// TIA Portal V18 export
VAR_GLOBAL   // PLC tag table "MemoryType"
   "PBB Off Mode" AT %M200.0 : Bool;
   "PBB On Mode" AT %M200.1 : Bool;
   "PBB Auto Mode" AT %M200.2 : Bool;
   "Emergency Stop Button Pressed" AT %M200.3 : Bool;
   "Tunnel FW Em Stop LS M" AT %M200.4 : Bool;
   "Tunnel BW Em Stop LS M" AT %M200.5 : Bool;
   "Start M" AT %M200.6 : Bool;
   "Fuse Problem Major" AT %M200.7 : Bool;
   "AutoLeveller Fault" AT %M201.0 : Bool;
   "AutoLeveller Up Over Work" AT %M201.1 : Bool;
   "AutoLeveller Down Over Work" AT %M201.2 : Bool;
   "Driver Error Left" AT %M201.3 : Bool;
   "Driver Error Right" AT %M201.4 : Bool;
   "Wheel Drivers Fault" AT %M201.5 : Bool;
   "SafetyShoe Siren&Info" AT %M201.6 : Bool;
   "SafetyBarrier Activated" AT %M201.7 : Bool;
   "Fault Occurred Major" AT %M202.1 : Bool;
   "Cabin Motor Driver Fault" AT %M202.2 : Bool;
   "Fault Occured Minor" AT %M202.3 : Bool;
   OK AT %M202.4 : Bool;
   "FW L1" AT %M202.5 : Bool;
   "FW L2" AT %M202.6 : Bool;
   "FW L3" AT %M202.7 : Bool;
   "BW L1" AT %M203.0 : Bool;
   "BW L2" AT %M203.1 : Bool;
   "BW L3" AT %M203.2 : Bool;
   "LFT L1" AT %M203.3 : Bool;
   "LFT L2" AT %M203.4 : Bool;
   "LFT L3" AT %M203.5 : Bool;
   "RGHT L1" AT %M203.6 : Bool;
   "RGHT L2" AT %M203.7 : Bool;
   "RGHT L3" AT %M204.0 : Bool;
   "JS Mid M" AT %M204.1 : Bool;
   "SafetyShoe Activated" AT %M204.2 : Bool;
   "AutoLeveller Up" AT %M204.3 : Bool;
   "AutoLeveller Down" AT %M204.4 : Bool;
   "sanal kesici (1)" AT %M204.5 : Bool;
   "Down Stop Object Limit" AT %M204.6 : Bool;
   "SafetyShoe Long Press" AT %M204.7 : Bool;
   "SS Cable Problem" AT %M205.0 : Bool;
   "AutoSafety Cross" AT %M205.1 : Bool;
   "AutoLeveller FW" AT %M205.2 : Bool;
   "AutoLeveller BW" AT %M205.3 : Bool;
   "Autoleveler temp count" AT %M205.4 : Bool;
   "Fuse Problem Minor" AT %M205.7 : Bool;
   "Wire Up Stop PBB" AT %M206.0 : Bool;
   "Slope Stop Up" AT %M206.1 : Bool;
   "Wire Up Stop PBB Limit All" AT %M206.2 : Bool;
   "Wire Down Stop PBB" AT %M206.3 : Bool;
   "Slope Stop Down" AT %M206.4 : Bool;
   "Down Stop Object" AT %M206.5 : Bool;
   "Down Stop PBB All" AT %M206.6 : Bool;
   "Speed L1" AT %IW100 : Int;
   "Speed L2" AT %IW102 : Int;
   "Speed L3" AT %IW104 : Int;
   "Slow Activated" AT %M207.2 : Bool;
   "Drive Slow Limit All" AT %M207.3 : Bool;
   "FW Slow Limit All" AT %M207.4 : Bool;
   "BW Slow Limit All" AT %M207.5 : Bool;
   "FW M" AT %M207.6 : Bool;
   "BW M" AT %M207.7 : Bool;
   "FW-LFT" AT %M208.0 : Bool;
   "FW-RGHT" AT %M208.1 : Bool;
   "BW-LFT" AT %M208.2 : Bool;
   "BW-RGHT" AT %M208.3 : Bool;
   "Cross M" AT %M208.4 : Bool;
   "FW Stop All" AT %M208.5 : Bool;
   "BW Stop All" AT %M208.6 : Bool;
   "LFT Stop All" AT %M208.7 : Bool;
   "RGHT Stop All" AT %M209.0 : Bool;
   "FW Allowed" AT %M209.1 : Bool;
   "BW Allowed" AT %M209.2 : Bool;
   "LFT Allowed" AT %M209.3 : Bool;
   "RGHT Allowed" AT %M209.4 : Bool;
   "FW-LFT Allowed" AT %M209.5 : Bool;
   "FW-RGHT Allowed" AT %M209.6 : Bool;
   "BW-LFT Allowed" AT %M209.7 : Bool;
   "BW-RGHT Allowed" AT %M210.0 : Bool;
   "Drive Angle Stop Left" AT %M210.1 : Bool;
   "Drive LSW Left Stop" AT %M210.2 : Bool;
   "Drive Angle Stop Right" AT %M210.3 : Bool;
   "Drive LSW Right Stop" AT %M210.4 : Bool;
   "Drive Slow Left Limit" AT %M210.5 : Bool;
   "Drive Slow Right Limit" AT %M210.6 : Bool;
   "Rotunda FW Stop LFT" AT %M210.7 : Bool;
   "Brake Off Time" AT %ID106 : Time;
   "Rotunda BW Stop LFT" AT %M211.0 : Bool;
   "Rotunda FW Stop RGHT" AT %M211.1 : Bool;
   "Rotunda BW Stop RGHT" AT %M211.2 : Bool;
   "Rotunda FW Stop All" AT %M211.3 : Bool;
   "Rotunda BW Stop All" AT %M211.4 : Bool;
   "Tunnel Laser FW Slow Limit" AT %M211.5 : Bool;
   "Tunnel LSW FW Slow" AT %M211.6 : Bool;
   "PhotoCell Slow Limit" AT %M211.7 : Bool;
   "UltraSonic Slow Limit" AT %M212.0 : Bool;
   "AirCraft Seen Anime" AT %M212.1 : Bool;
   "Laser BW Slow Limit" AT %M212.2 : Bool;
   "LS BW Slow Limit" AT %M212.3 : Bool;
   "Laser FW Stop Limit" AT %M212.5 : Bool;
   "LS FW Stop Limit" AT %M212.7 : Bool;
   "Touch LFT Stop Limit" AT %M213.0 : Bool;
   "Touch Mid Stop Limit" AT %M213.1 : Bool;
   "Touch RGTH Stop Limit" AT %M213.2 : Bool;
   "AirCraft Touch Anime" AT %M213.3 : Bool;
   "Laser BW Stop Limit" AT %M213.4 : Bool;
   "LS BW Stop Limit" AT %M213.5 : Bool;
   "FW G120C Stop" AT %M213.7 : Bool;
   "BW G120C Stop" AT %M214.0 : Bool;
   "LFT G120C Stop" AT %M214.1 : Bool;
   "Right G120C Stop" AT %M214.2 : Bool;
   "FW-LFT G120C Stop" AT %M214.3 : Bool;
   "FW-RGHT G120C Stop" AT %M214.4 : Bool;
   "BW-LFT G120C Stop" AT %M214.5 : Bool;
   "BW-RGHT G120C Stop" AT %M214.6 : Bool;
   "Cab Angle Left Stop" AT %M214.7 : Bool;
   "Cab LS Left Stop" AT %M215.0 : Bool;
   "Cab Stop Left All" AT %M215.1 : Bool;
   "Cab Angle Right Stop" AT %M215.2 : Bool;
   "Cab LS Right Stop" AT %M215.3 : Bool;
   "Cab Stop Right All" AT %M215.4 : Bool;
   "Rotunda Stop Angle Rght" AT %M215.5 : Bool;
   "Rotunda Stop Angle LFT" AT %M215.6 : Bool;
   "Canopy BW Auto" AT %M216.0 : Bool;
   "canopy ok1" AT %M216.1 : Bool;
   "canopy ok2" AT %M216.2 : Bool;
   memo2 AT %M216.3 : Bool;
   memo AT %M216.4 : Bool;
   memo3 AT %M216.5 : Bool;
   memo4 AT %M220.0 : Bool;
   "SE ByPass" AT %M220.2 : Bool;
   "Tunnel Real Meter" AT %MD300 : Real;
   "Drive Angle Real Meter" AT %MD304 : Real;
   "Rotunda Angle Real Meter" AT %MD312 : Real;
   "Height Real" AT %MD332 : Real;
   "Cab Angle Real Meter" AT %MD348 : Real;
   "Rotunda Stop LS LFT" AT %M216.6 : Bool;
   "Rotunda Stop LS Rght" AT %M225.5 : Bool;
   "Slope Angel" AT %MD615 : Real;
   "Slope Vertical" AT %MD620 : Real;
   "Slope Stop All" AT %M225.6 : Bool;
   "Speed Active L1" AT %M225.7 : Bool;
   "Speed Active L2" AT %M226.2 : Bool;
   "Speed Active L3" AT %M226.3 : Bool;
   "Rotunda Slow Angle Rght" AT %M215.7 : Bool;
   "Rotunda Slow Angle LFT" AT %M216.7 : Bool;
   "Rotunda Slow Angle ALL" AT %M217.6 : Bool;
   "Slope Slow Down" AT %M206.7 : Bool;
   "Slope Slow Up" AT %M207.0 : Bool;
   "Slope Slow ALL" AT %M207.1 : Bool;
   "Fast Mode" AT %M226.0 : Bool;
   "Service GPU Active" AT %M202.0 : Bool;
   "Service PCA Active" AT %M205.5 : Bool;
   "Service Hose Active" AT %M205.6 : Bool;
   "Service Air Active" AT %M212.4 : Bool;
   "Drive Angle LS FW Stop" AT %M212.6 : Bool;
   "Drive Angle LS BW Stop" AT %M213.6 : Bool;
   "R6 - Cab Warning Light & Buzzer Test" AT %M226.4 : Bool;
END_VAR
